PROGRAM PrincipalClient2
VAR
	facade1 : FacadePrinterNormal(text:= 'text 1', color:= TRUE , sheet:= 'A1', documentType:='PDF');
         
    facade2 : FacadePrinterNormal(text:= 'text 2', color:= FALSE , sheet:= 'A2', documentType:='Excel');
	                  
    i3 : printer;
	
	startdemo : BOOL;
	
END_VAR


IF  startdemo THEN
	
	startdemo := FALSE;

	facade1.print();
			
	facade2.print();
			 
	i3.setSheet('A3');
    i3.setColor(TRUE);
    i3.setDocumenttype('RTF');
    i3.setText('text 3');
    i3.printDocument();
	
END_IF

END_PROGRAM

(* stored: Version 1.1.0.1, ProductVersion 3.1.4024.12
   POU PrincipalClient2: Id {b5e7a9bb-5c42-41eb-8b4d-222ead27472d}, SpecialFunc None *)
